// TIA Portal V16 export
// export: Created 2020-12-17T10:24:08.949615Z, ExportSetting WithDefaults, DisplayName Totally Integrated Automation Portal, DisplayVersion V16 Update 2, DisplayName TIA Portal Version Control Interface, DisplayVersion V16 Update 2, DisplayName TIA Portal Openness, DisplayVersion V16 Update 2, DisplayName STEP 7 Professional, DisplayVersion V16 Update 2, DisplayName STEP 7 Safety, DisplayVersion V16, DisplayName WinCC Advanced / Unified PC, DisplayVersion V16 Update 2
ORGANIZATION_BLOCK "Main"   // OB1, LAD, ProgramCycle
TITLE = "Main Program Sweep (Cycle)"
{ S7_Optimized_Access := 'TRUE' }
VERSION : 0.1
// stored: AutoNumber true, IsIECCheckEnabled false, SetENOAutomatically false
   VAR_INPUT
      Initial_Call : Bool;   // Initial call of this OB
      Remanence : Bool;   // =True, if remanent data are available
   END_VAR
BEGIN

REGION Network 1
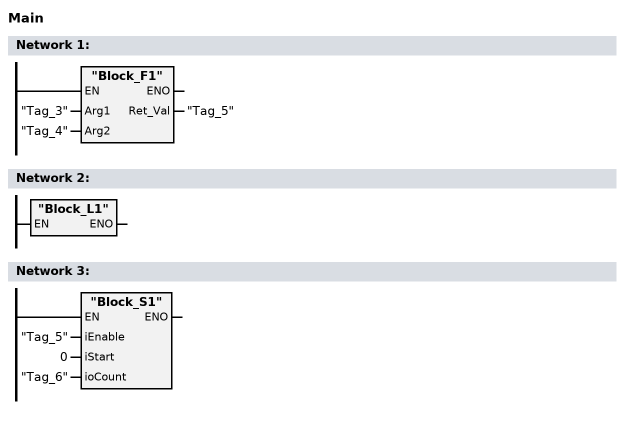
   RUNG wire#powerrail
      "Block_F1"(Arg1 := "Tag_3", Arg2 := "Tag_4", Ret_Val => "Tag_5")
   END_RUNG
   // the same network as SCL:
   "Tag_5" := "Block_F1"(Arg1 := "Tag_3", Arg2 := "Tag_4");
END_REGION

REGION Network 2
   RUNG wire#powerrail
      "Block_L1"()
   END_RUNG
   // the same network as SCL:
   "Block_L1"();
END_REGION

REGION Network 3
   RUNG wire#powerrail
      "Block_S1"(iEnable := "Tag_5", iStart := 0, ioCount := "Tag_6")
   END_RUNG
   // the same network as SCL:
   "Block_S1"(iEnable := "Tag_5", iStart := 0, ioCount := "Tag_6");
END_REGION
END_ORGANIZATION_BLOCK
